FUNCTION_BLOCK FB_PumpGrundfosMagna3 EXTENDS FB_ActorContinous
VAR_INPUT
	nControlModeAutomatic : E_GrundfosMagna3ControlMode; //Grundfos Magna3 control modes
	fExternalValue : REAL; //external value for control, e. g. temperature, temperature difference volume flow rate
END_VAR
VAR_OUTPUT
	bError : BOOL; //true if pump is in error
	fTemperatureInternal : REAL; //internal temperature (e.g. for temperature controlling valves)
	fTemperatureExternal : REAL; //external temperature (e.g. for temperature controlling valves)
END_VAR
VAR
	{attribute 'OPC.UA.DA' := '1'}
	localSetParameters : ST_PumpGrundfosMagna3SetParameters;
	{attribute 'OPC.UA.DA' := '1'}
	localState : ST_PumpGrundfosMagna3State;
	
	//default parameters
	localDefaultParameters : ST_PumpGrundfosMagna3DefaultParameters;
	
	//I/O links
	StatusModule_IN				AT %I* : ARRAY [0..5] OF BYTE;
	nAlarmCode_IN				AT %I* : USINT;
	nWarningCode_IN				AT %I* : USINT;
	fVolumeFlowRate_IN 			AT %I* : UDINT; //m^3/h volume flow rate from pump
	fPressureDifference_IN	 	AT %I* : UDINT; //pa = 10^-5 bar
	fPowerElectric_IN			AT %I* : UDINT; //W
	fTemperatureInternal_IN 	AT %I* : REAL; //°C
	fActualSetpoint_IN			AT %I* : UDINT; //%
	fRotationalSpeed_IN	 		AT %I* : UDINT; //rpm
	fTemperatureExternal_IN 	AT %I* : UDINT; //°C external temperature from sensor connected to pump
	fTemperatureDifference_IN	AT %I* : UDINT; //°C
	fPowerThermal_IN	 		AT %I* : UDINT; //W
	ControlModule_OUT 			AT %Q* : ARRAY [0..4] OF BYTE;
	
	//controllers
	PI_Controller				: FB_CTRL_PI; 
	PI_Controller_Parameters 	: ST_CTRL_PI_PARAMS;
	fSetpointValue : LREAL; //internal setpoint value (is switched depending on heating/cooling application)
	fActualValue : LREAL; //internal setpoint value (is switched depending on heating/cooling application)
	fAct : REAL; //actual measured value from internal pump sensor or external sensor
		
	//internal variables:
	nControlMode : E_GrundfosMagna3ControlMode; //actual pump control mode
	fSetPoint_controlled : REAL; //controlled setpoint
END_VAR

MAIN();
SelectPumpControlMode();
CalculateHydraulicPower();
ControlPump();

METHOD PRIVATE CalculateHydraulicPower : REAL
VAR_INPUT
END_VAR
localState.fPowerHydraulic := localState.fPressureDifference*localState.fVolumeFlowRate;
END_METHOD

METHOD PRIVATE ControlPump : BOOL
VAR_INPUT
END_VAR
VAR
END_VAR
//set control parameters
PI_Controller_Parameters.fKp 				:= localDefaultParameters.fControllerAmplification;
PI_Controller_Parameters.tTn 				:= localDefaultParameters.tControllerIntegralTime;
PI_Controller_Parameters.fOutMaxLimit		:= 100.0;
PI_Controller_Parameters.fOutMinLimit		:= 0.0;
PI_Controller_Parameters.tTaskCycleTime		:= localDefaultParameters.tTaskCycleTime;
PI_Controller_Parameters.tCtrlCycleTime		:= localDefaultParameters.tCtrlCycleTime;
PI_Controller_Parameters.bARWOnIPartOnly	:= TRUE;

//check which actual value should be used depending on control mode, external temperature sensor and pump place
CASE nControlMode OF
	1,2: //constant temperature control
	IF localDefaultParameters.bPumpBeforeApplication THEN
		IF localDefaultParameters.bExternalTemperatureSensor THEN
			fAct := localState.fTemperatureExternal;
		ELSE
			fAct := fExternalValue;
		END_IF
	ELSE
		fAct := localState.fTemperatureInternal;		
	END_IF
	3: //temperature difference control
	fAct := localState.fTemperatureDifference;
	IF localDefaultParameters.bPumpBeforeApplication AND NOT localDefaultParameters.bExternalTemperatureSensor THEN
		fAct := fExternalValue;
	END_IF
END_CASE

//switch setpoint and actual value depending on heating or cooling mode
CASE nControlMode OF
	1: //flow is heated
	fSetpointValue := fAct;
	fActualValue := fSetPoint;	

	2: //flow is cooled
	fSetpointValue := fSetPoint;	
	fActualValue := fAct;
	
	3: //temperature difference
	fSetpointValue := ABS(fAct);
	fActualValue := ABS(fSetPoint);
END_CASE

PI_Controller (
		fSetpointValue	:= fSetpointValue,
		fActualValue	:= fActualValue,
		fManSyncValue	:= 0,
		bSync			:= FALSE,
		eMode			:= 2, (* mode active *)
		bHold			:= FALSE,
		stParams		:= PI_Controller_Parameters);

//output of PI controller is not used in frequency control mode
CASE nControlMode OF
	0:
	fSetPoint_controlled := fSetPoint;
ELSE	
	fSetPoint_controlled := LREAL_TO_REAL(PI_Controller.fOut);
END_CASE
END_METHOD

METHOD GetState_Profibus : BOOL
VAR_INPUT
END_VAR
VAR
	controlModule0Bits : ARRAY[0..7] OF BOOL;
END_VAR
controlModule0Bits := ConvertByteToBit(dataByte:=StatusModule_IN[0]);

//control state
controlState.bStatusOn := controlModule0Bits[1];
bSetStatusOn := controlState.bStatusOn;

//setpoint state
setPointState.fOperatingPoint := BufferUdintToReal(raw_input := fActualSetpoint_IN);
fOperatingPoint := setPointState.fOperatingPoint;
setPointState.sOperatingPointUnit := 'percent';

//local state
localState.bError := controlModule0Bits[2];
localState.bWarning := controlModule0Bits[3];
bError := localState.bError;
localState.sErrorMessage := CONCAT('Alarm code: ',INT_TO_STRING(nAlarmCode_IN));
localState.sWarningMessage := CONCAT('Warning code: ',INT_TO_STRING(nWarningCode_IN));
localState.bRemoteControlOn := controlModule0Bits[0];
localState.fVolumeFlowRate := BufferUdintToReal(raw_input := fVolumeFlowRate_IN);
localState.fTemperatureInternal := BufferRealToReal(raw_input := fTemperatureInternal_IN);
fTemperatureInternal := localState.fTemperatureInternal;
IF localDefaultParameters.bExternalTemperatureSensor THEN //Set external temperature and temperature difference if temperature sensor is connected
	localState.fTemperatureExternal := BufferUdintToReal(raw_input := fTemperatureExternal_IN);
	fTemperatureExternal := localState.fTemperatureExternal;
	localState.fTemperatureDifference := BufferUdintToReal(raw_input := fPressureDifference_IN);
END_IF;
localState.fPressureDifference := BufferUdintToReal(raw_input := fPressureDifference_IN);
localState.fPowerElectric := BufferUdintToReal(raw_input := fPowerElectric_IN);
localState.fPowerThermal := BufferUdintToReal(raw_input := fPowerThermal_IN);
localState.fRotationalSpeed := BufferUdintToReal(raw_input := fRotationalSpeed_IN);
END_METHOD

METHOD PRIVATE SelectPumpControlMode : BOOL
VAR_INPUT
END_VAR
IF control.bManualModeActivated THEN
	nControlMode := localSetParameters.nControlModeManual;
ELSIF control.bAlgorithmModeActivated AND bAlgorithmPermission THEN
	nControlMode := localSetParameters.nControlModeAlgorithm;
ELSE
	nControlMode := nControlModeAutomatic;
END_IF
END_METHOD

METHOD PROTECTED  SetSetPointLimits : BOOL
VAR_INPUT
END_VAR
aSetPointLimits := localDefaultParameters.aSetPointLimits;
END_METHOD

METHOD SetState_Profibus : BOOL
VAR_INPUT
END_VAR
VAR
	tmp : STRING;
	controlModule0Bits : ARRAY[0..7] OF BOOL;
END_VAR
//setpoint state
setPointState.fSetPoint := fSetPoint;
setPointState.aSetPointLimits := aSetPointLimits;
CASE nControlMode OF
	0: //position mode
	setPointState.sSetPointUnit := 'percent';
	
	1,2: //constant temperature
	setPointState.sSetPointUnit := 'degreeC';
	
	3: //temperature difference
	setPointState.sSetPointUnit := 'K';
END_CASE

//output
controlModule0Bits[0] := TRUE; //Remote control
controlModule0Bits[1] := bSetStatusOn;//bit for switching on pump
controlModule0Bits[2] := localSetParameters.bReset; //bit to reset errors and warnings

ControlModule_OUT[0] := ConvertBitToByte(dataBit:=controlModule0Bits);
ControlModule_OUT[1] := 1;
ControlModule_OUT[2] := 0;
tmp := DWORD_TO_HEXSTR(DINT_TO_DWORD(TRUNC(fSetPoint_controlled*100)),4,TRUE);
ControlModule_OUT[3] := HEXCHRNIBBLE_TO_BYTE(MID(tmp,1,1))*16 + HEXCHRNIBBLE_TO_BYTE(MID(tmp,1,2));
ControlModule_OUT[4] := HEXCHRNIBBLE_TO_BYTE(MID(tmp,1,3))*16 + HEXCHRNIBBLE_TO_BYTE(MID(tmp,1,4));
END_METHOD

PROPERTY ST_DefaultParameters : REFERENCE TO ST_PumpGrundfosMagna3DefaultParameters
SET
localDefaultParameters := ST_DefaultParameters;
END_SET
END_PROPERTY

END_FUNCTION_BLOCK

(* stored: Version 1.1.0.1, ProductVersion 3.1.4024.10
   POU FB_PumpGrundfosMagna3: Id {5ff4732a-f57a-4b28-83eb-fee6b9ba074e}, SpecialFunc None
   Method CalculateHydraulicPower: Id {5ee59af5-7c08-4f03-8cfe-829337b66dfd}
   Method ControlPump: Id {812b0398-87f0-4a15-8dd7-9c34771d439d}
   Method GetState_Profibus: Id {14b06936-b53d-4b61-8427-f5bf98ac63d6}
   Method SelectPumpControlMode: Id {9f36f1dc-61c9-4f36-814e-95f20eaaf659}
   Method SetSetPointLimits: Id {98846448-9692-42fd-b02a-6804c1f2306d}
   Method SetState_Profibus: Id {26cf015c-036e-449a-a37e-24bce7fc2f85}
   Property ST_DefaultParameters: Id {37c47602-10af-4f25-93f4-2c0dd2131db3}
   Set Set: Id {69ad99eb-9ef1-4940-bed0-9eace3e8cb70} *)
